// Mitsubishi GX Works2 project: LOS   PLC: FX3U/FX3UC

PROGRAM MAIN
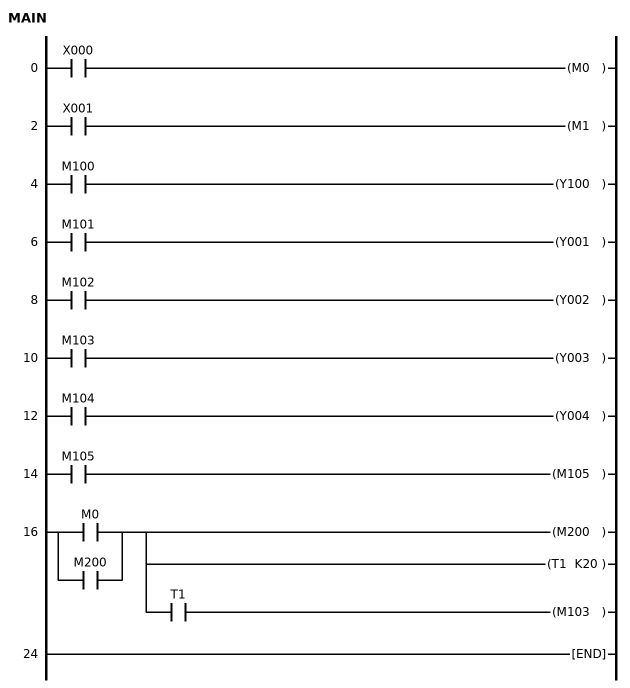
0     LD      X000
      OUT     M0
2     LD      X001
      OUT     M1
4     LD      M100
      OUT     Y100
6     LD      M101
      OUT     Y001
8     LD      M102
      OUT     Y002
10    LD      M103
      OUT     Y003
12    LD      M104
      OUT     Y004
14    LD      M105
      OUT     M105
16    LD      M0
      OR      M200
      OUT     M200
      OUT     T1 K20
      AND     T1
      OUT     M103
24    END
END_PROGRAM
